FUNCTION_BLOCK XtsProcessingUnitControl
VAR_INPUT
END_VAR
VAR_OUTPUT
END_VAR
VAR	
	
	LocalState				: BYTE;
	DetectedMoverCount		: UDINT;
	ActiveMoverCount		: UDINT;
	ScannedModuleCount		: UDINT;
	DriveState				: DriveState;
	AxisID					: UDINT;
	MoverIdDetectionDone	: BOOL;
	Initialized				: BOOL;
	
	Environment				: FB_TcIoXtsEnvironment;
	EnvironmentConfig		: ST_XtsEnvironmentConfiguration;
	ProcessingUnit			: FB_TcIoXtsProcessingUnit;
	InfoServer				: FB_TcIoXtsInfoServer;
	InfoServerAndStation	: FB_TcIoXtsInfoServerInfoStation;
	CaGroup					: FB_Mc2CaGroup;

	XpuPart					: FB_TcIoXtsXpuPart;
	PartModule				: FB_TcIoXtsPartModule;
	PartControlArea			: FB_TcIoXtsPartControlArea;
	XpuTrack				: FB_TcIoXtsXpuTrack;
	XpuMover				: FB_TcIoXtsXpuMover;
	
END_VAR

// NETWORK 1

METHOD CyclicUpdate : BOOL
VAR_INPUT
	nXpu		: UINT;
END_VAR
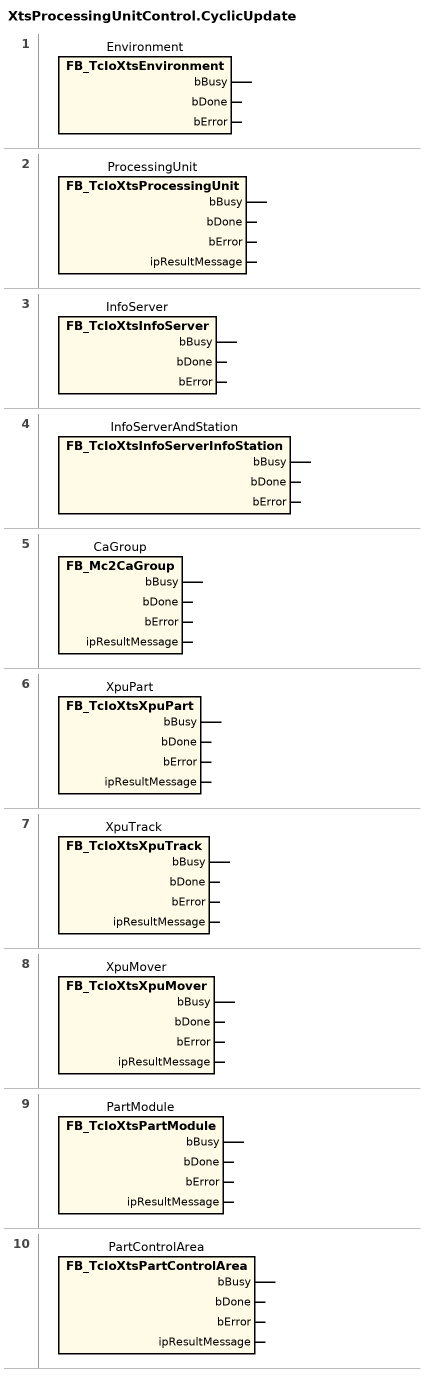
// NETWORK 1
Environment(); // FB_TcIoXtsEnvironment

// NETWORK 2
ProcessingUnit(); // FB_TcIoXtsProcessingUnit

// NETWORK 3
InfoServer(); // FB_TcIoXtsInfoServer

// NETWORK 4
InfoServerAndStation(); // FB_TcIoXtsInfoServerInfoStation

// NETWORK 5
CaGroup(); // FB_Mc2CaGroup

// NETWORK 6
XpuPart(); // FB_TcIoXtsXpuPart

// NETWORK 7
XpuTrack(); // FB_TcIoXtsXpuTrack

// NETWORK 8
XpuMover(); // FB_TcIoXtsXpuMover

// NETWORK 9
PartModule(); // FB_TcIoXtsPartModule

// NETWORK 10
PartControlArea(); // FB_TcIoXtsPartControlArea

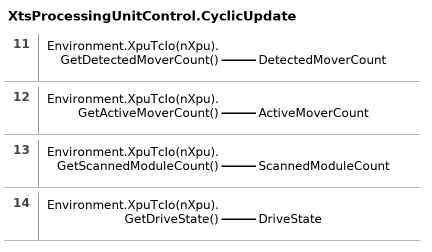
// NETWORK 11
DetectedMoverCount := Environment.XpuTcIo(nXpu).GetDetectedMoverCount();

// NETWORK 12
ActiveMoverCount := Environment.XpuTcIo(nXpu).GetActiveMoverCount();

// NETWORK 13
ScannedModuleCount := Environment.XpuTcIo(nXpu).GetScannedModuleCount();

// NETWORK 14
DriveState := Environment.XpuTcIo(nXpu).GetDriveState();
END_METHOD

METHOD Initialize : BOOL
VAR_INPUT
END_VAR

// Call once to configure the XTS environment

CASE LocalState OF

	0:
		EnvironmentConfig.bEnableInitInfoServer := TRUE;
		EnvironmentConfig.bEnableInitCaGroup := TRUE;
		Environment.P_XtsEnvironmentConfiguration := EnvironmentConfig;
		LocalState := 1;
		
	1:
		IF Environment.Init(TRUE) THEN
			Environment.Init(FALSE);
			LocalState := 2;
		END_IF
		
	2:
		IF Environment.P_IsInitialized THEN
			Initialized := TRUE;
			LocalState := 3;
		END_IF
		
	3:
		IF Environment.XpuTcIo(1).SetMoverIdDetectionMode(MoverIdDetectionMode.Mover1) THEN
			LocalState := 4;
		END_IF
		
	4:
		IF Environment.XpuTcIo(1).TriggerMoverIdDetection() THEN
			MoverIdDetectionDone := TRUE;
			LocalState := 5;
		END_IF
		
	5:
		LocalState := 0;
		Initialize := TRUE;	
		
END_CASE
END_METHOD

END_FUNCTION_BLOCK

(* stored: Version 1.1.0.1, ProductVersion 3.1.4024.12
   POU XtsProcessingUnitControl: Id {686c9d06-3079-48b0-9c02-90d015e45ce4}, SpecialFunc None
   Folder Power and Utility: Id {57efb649-b87b-4146-95c4-7b48f473b0a4}
   Method CyclicUpdate: Id {04ce8273-f602-4fb5-b977-7e0b2f719e39}
   Method Initialize: Id {3ad1bebe-74e4-4508-8b52-780a319c2d96} *)
